// TIA Portal V17 export
// export: Created 2025-01-08T13:55:35.8985116Z, ExportSetting WithDefaults, DisplayName Totally Integrated Automation Portal, DisplayVersion V17, DisplayName TIA Portal Openness, DisplayVersion V17, DisplayName TIA Portal Version Control Interface, DisplayVersion V17, DisplayName SINAMICS Startdrive Advanced, DisplayVersion V17 Update2, DisplayName SINAMICS Startdrive G130, G150, S120, S150, SINAMICS MV, S210, DisplayVersion V17 Update2, DisplayName SINAMICS Startdrive G110M, G120, G120C, G120D, G120P, G115D, DisplayVersion V17 Update2, DisplayName STEP 7 Professional, DisplayVersion V17, DisplayName STEP 7 Safety, DisplayVersion V17, DisplayName WinCC Advanced, DisplayVersion V17
VAR_GLOBAL   // PLC tag table "Default tag table"
   System_Byte AT %MB1000 : Byte;
   FirstScan AT %M1000.0 : Bool;
   DiagStatusUpdate AT %M1000.1 : Bool;
   AlwaysTRUE AT %M1000.2 : Bool;
   AlwaysFALSE AT %M1000.3 : Bool;
   Clock_Byte AT %MB1001 : Byte;
   Clock_10Hz AT %M1001.0 : Bool;
   Clock_5Hz AT %M1001.1 : Bool;
   "Clock_2.5Hz" AT %M1001.2 : Bool;
   Clock_2Hz AT %M1001.3 : Bool;
   "Clock_1.25Hz" AT %M1001.4 : Bool;
   Clock_1Hz AT %M1001.5 : Bool;
   "Clock_0.625Hz" AT %M1001.6 : Bool;
   "Clock_0.5Hz" AT %M1001.7 : Bool;
   TestReceive AT %M0.0 : Bool;
   ProductIn_Mem AT %M2.0 : LInt;
   GitTest AT %M0.1 : Bool;
END_VAR
